TYPE (* A Structure with 16 Bits *)
  (* Version 1.0, 2024-02-21, franz *)
  st16b : STRUCT
    b00 : BOOL; (* BIT 00 *)
    b01 : BOOL; (* BIT 01 *)
    b02 : BOOL; (* BIT 02 *)
    b03 : BOOL; (* BIT 03 *)
    b04 : BOOL; (* BIT 04 *)
    b05 : BOOL; (* BIT 05 *)
    b06 : BOOL; (* BIT 06 *)
    b07 : BOOL; (* BIT 07 *)
    b08 : BOOL;
    b09 : BOOL;
    b10 : BOOL;
    b11 : BOOL;
    b12 : BOOL;
    b13 : BOOL;
    b14 : BOOL;
    b15 : BOOL;
  END_STRUCT;
END_TYPE
